{attribute 'GeneratedUsingTerminal: EM3702-0000-0016'}
{attribute addProperty BoxType "EM3702-0000-0016"}
{attribute addProperty Id "StatusAT %I*Status_E3F6A94B6ValueAT %I*INT2"}
{attribute addProperty CRC "1526095950"}
{attribute addProperty Size "8"}
TYPE AI_Input_Channel_5AF6604E EXTENDS InputBase_8311D824 :
STRUCT
	{attribute addProperty Name "Status"}
	Status AT %I* : Status_E3F6A94B;
	{attribute addProperty Name "Value"}
	Value AT %I* : INT;
END_STRUCT
END_TYPE

(* stored: Version 1.2.0.0, ProductVersion 3.1.4024.9
   DUT AI_Input_Channel_5AF6604E: Id {a6df6835-c37e-41ab-a1a4-f8b1df1bf366} *)
